(* CoDeSys 2.3 export: MonitorBool.EXP *)

(* POU basic/MonitorBool, ST *)
FUNCTION MonitorBool : BOOL
VAR_INPUT
    Group: BYTE;
    Id: BYTE;
    Channel: UINT;
    Value: BOOL;
END_VAR
VAR_IN_OUT
    Data: BOOL;
END_VAR
VAR
END_VAR
IF Value <> Data THEN
    IF Group > 0 OR Id > 0 THEN
        IF Channel < 256 THEN
            EvtGr8Id8Ch8Tick32Bool8(Group, Id, UINT_TO_BYTE(Channel), GlobalTick, Value, GlobalLogBufferHandle);
        ELSE
            EvtGr8Id8Ch16Tick32Bool8(Group, Id, Channel, GlobalTick, Value, GlobalLogBufferHandle);
        END_IF
    ELSIF Channel < 256 THEN
        EvtCh8Tick32Bool8(UINT_TO_BYTE(Channel), GlobalTick, Value, GlobalLogBufferHandle);
    ELSE
        EvtCh16Tick32Bool8(Channel, GlobalTick, Value, GlobalLogBufferHandle);
    END_IF
    Data := Value;
END_IF
END_FUNCTION
